// SIMATIC S7-200 SMART project (STEP 7-Micro/WIN SMART), CPU SR40

SYMBOL_TABLE 用户定义1
运算结果             VD20
END_SYMBOL_TABLE

ORGANIZATION_BLOCK 主程序:OB1
TITLE=程序注释
BEGIN
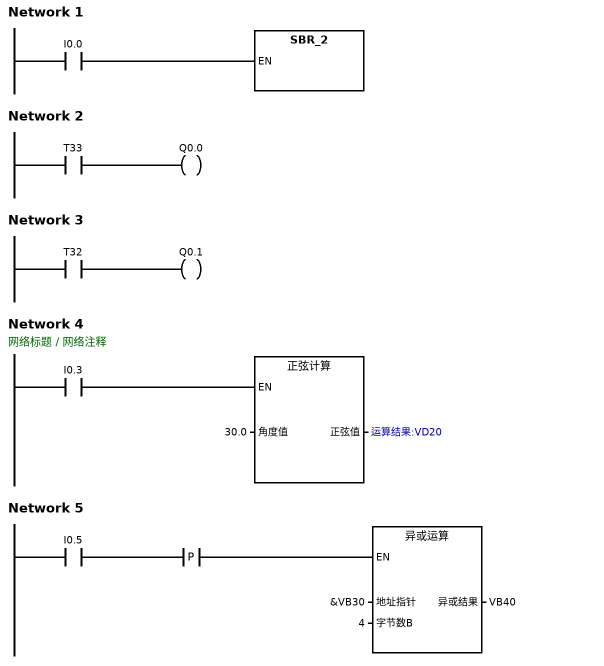
Network 1
LD     I0.0
CALL   SBR_2:SBR2
Network 2
LD     T33
=      Q0.0
Network 3
LD     T32
=      Q0.1
Network 4
// 网络标题
// 网络注释
LD     I0.3
CALL   正弦计算:SBR0, 30.0, 运算结果:VD20
Network 5
LD     I0.5
EU
CALL   异或运算:SBR1, &VB30, 4, VB40
END_ORGANIZATION_BLOCK

SUBROUTINE_BLOCK 正弦计算:SBR0
TITLE=子程序注释
VAR_INPUT
角度值:REAL;	// LD0 
END_VAR
VAR_OUTPUT
正弦值:REAL;	// LD4 
END_VAR
VAR
弧度值:REAL;	// LD8 
END_VAR
BEGIN
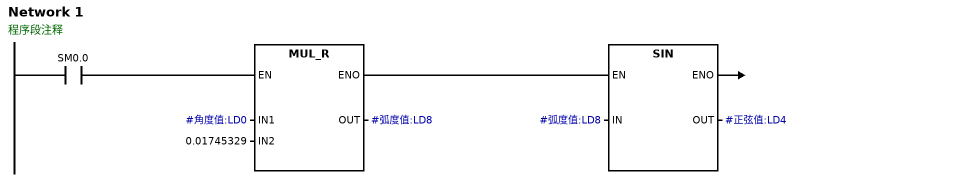
Network 1
// 程序段注释
LD     SM0.0
MOVR   #角度值:LD0, #弧度值:LD8
AENO
*R     0.01745329, #弧度值:LD8
AENO
SIN    #弧度值:LD8, #正弦值:LD4
END_SUBROUTINE_BLOCK

SUBROUTINE_BLOCK 异或运算:SBR1
TITLE=子程序注释
VAR_INPUT
地址指针:DWORD;	// LD0 
字节数B:BYTE;	// LB4 
END_VAR
VAR_OUTPUT
异或结果:BYTE;	// LB5 
END_VAR
VAR
循环计数器:INT;	// LW6 
字节数I:INT;	// LW8 
END_VAR
BEGIN
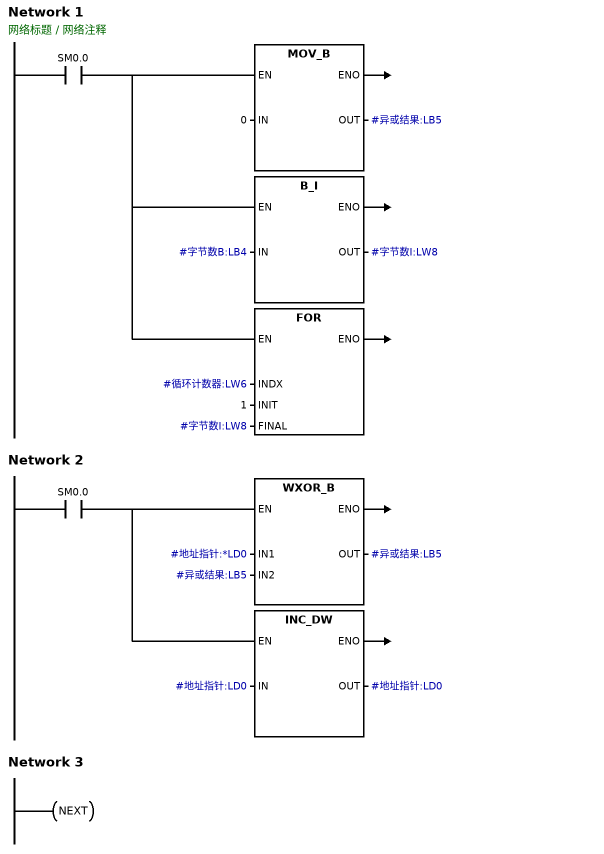
Network 1
// 网络标题
// 网络注释
LD     SM0.0
MOVB   0, #异或结果:LB5
BTI    #字节数B:LB4, #字节数I:LW8
FOR    #循环计数器:LW6, 1, #字节数I:LW8
Network 2
LD     SM0.0
XORB   *#地址指针:LD0, #异或结果:LB5
INCD   #地址指针:LD0
Network 3
NEXT
END_SUBROUTINE_BLOCK

SUBROUTINE_BLOCK SBR_2:SBR2
TITLE=子例程注释
BEGIN
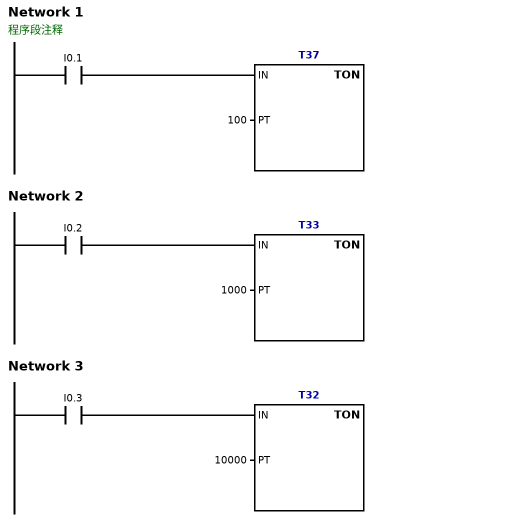
Network 1
// 程序段注释
LD     I0.1
TON    T37, 100
Network 2
LD     I0.2
TON    T33, 1000
Network 3
LD     I0.3
TON    T32, 10000
END_SUBROUTINE_BLOCK
